// TIA Portal V20 export
FUNCTION_BLOCK "FB_Sensors"   // FB16, LAD
{ S7_Optimized_Access := 'TRUE' }
// stored: MemoryReserve 100, SetENOAutomatically false
   VAR
      instDeviceSensor_010BX1 { S7_SetPoint := 'True'} : "deviceSensor";
   END_VAR
BEGIN

REGION Network 1: ----- FILTER -----
END_REGION

REGION Network 2: Sensor 1 Ind.s. (30BX1)
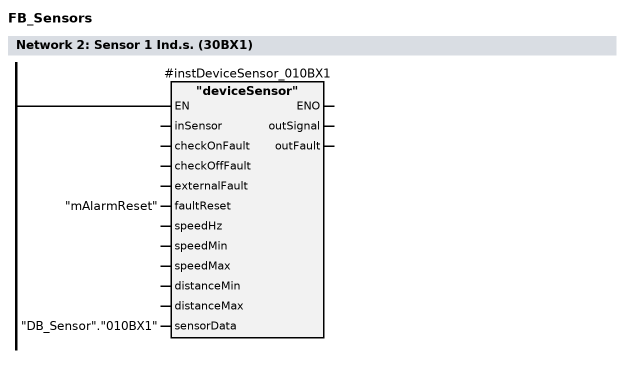
   RUNG wire#powerrail
      #instDeviceSensor_010BX1(inSensor :=, checkOnFault :=, checkOffFault :=, externalFault :=, faultReset := "mAlarmReset", speedHz :=, speedMin :=, speedMax :=, distanceMin :=, distanceMax :=, sensorData := "DB_Sensor"."010BX1", outSignal =>, outFault =>)
   END_RUNG
   // the same network as SCL:
   #instDeviceSensor_010BX1(faultReset := "mAlarmReset", sensorData := "DB_Sensor"."010BX1");   // "deviceSensor"
END_REGION
END_FUNCTION_BLOCK
